TYPE
    CU00xTechnologicalData EXTENDS TcoCore.TcoStruct : 
    STRUCT		
        
    END_STRUCT
END_TYPE

(* stored: Version 1.1.0.1
   DUT CU00xTechnologicalData: Id {d95b8f9e-2371-030e-0483-bd2dc1a02cc1} *)
